TYPE "MachineStatus"
VERSION : 0.1
// Block: MachineStatus
   STRUCT
      AtLeastOneMachineIsAborting : Bool;
      AllMachineAutReady : Bool;
      AllMachineAckStopInPhase : Bool;
      AllMachineAckStopProgrammed : Bool;
      AtLeastOneWngPresence : Bool;
      AtLeastOneAlrPresence : Bool;
   END_STRUCT;

END_TYPE
